{attribute 'qualified_only'}
{attribute 'strict'}
TYPE E_CoEParamState :
(
    eInit := -2,
    eReadName := -1,
    eIdle := 0,
    eWriteStart := 1,
    eWriteWaitingForDone := 2,
    eReadDriveParam := 11,
    eError := 100
);
END_TYPE

(* stored: Version 1.1.0.1
   DUT E_CoEParamState: Id {7b256909-45ff-4fb5-8610-f99052702492} *)
